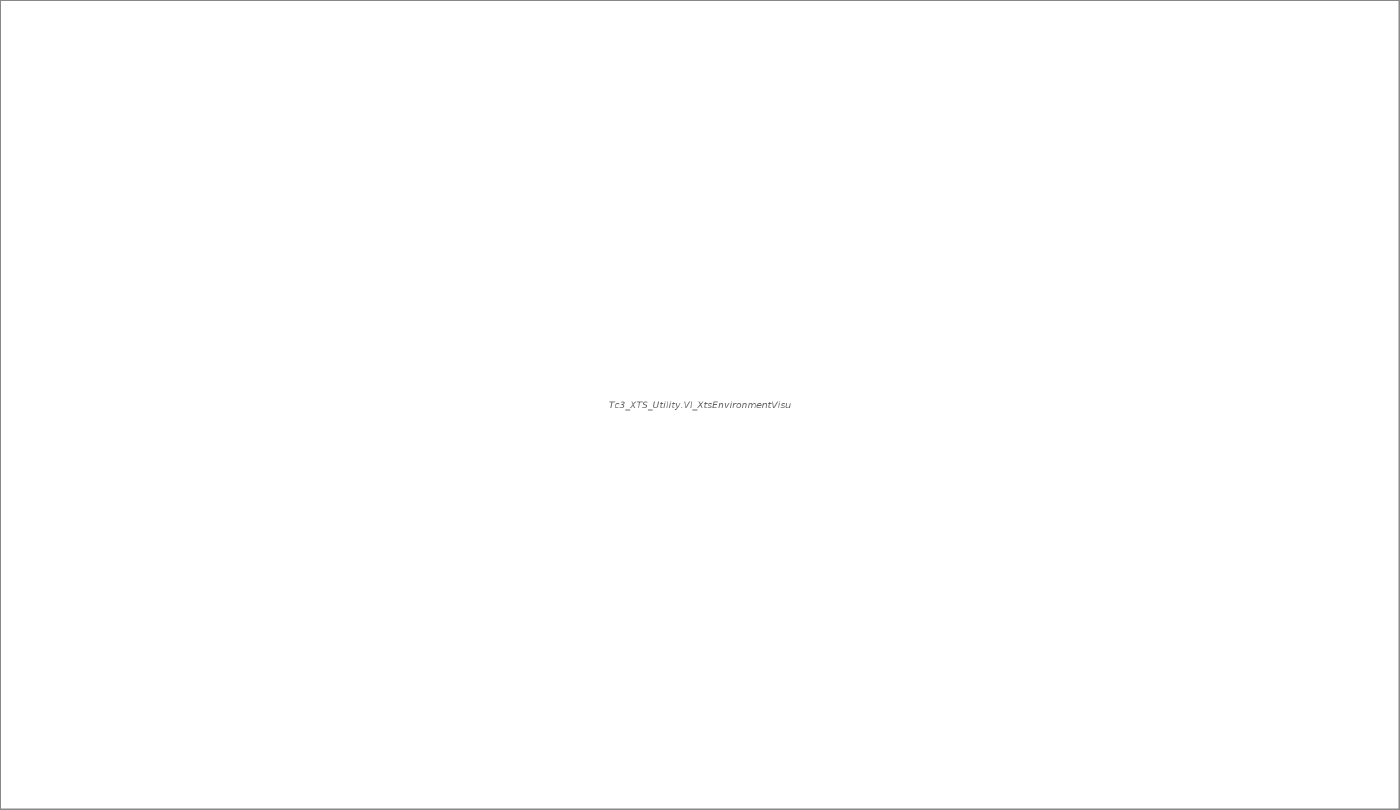
VISUALIZATION PageXtsEnviroment_1  // 1520x880
    Frame (0,0 1520x880)
        shows Tc3_XTS_Utility.VI_XtsEnvironmentVisu()
END_VISUALIZATION

(* stored: Version 1.1.0.1, ProductVersion 3.1.4024.12
   Visu PageXtsEnviroment_1: Id {3c1716ae-968c-417e-ac4a-e30b8bfc4bb6} *)
